FUNCTION_BLOCK KukaRobot
VAR_INPUT
END_VAR
VAR
	wSendData : DWORD;
END_VAR
VAR_OUTPUT
	wOutputWord AT %Q* : DWORD;
END_VAR

METHOD SendData : BOOL
VAR_INPUT
	bFailure : BOOL := FALSE;
END_VAR
IF bFailure THEN
	wOutputWord := 16#00000001;
ELSE
	wOutputWord:= 16#00000000;
END_IF
END_METHOD

END_FUNCTION_BLOCK

(* stored: Version 1.1.0.1, ProductVersion 3.1.4024.12
   POU KukaRobot: Id {468c34ef-d238-4a9f-8ae3-3cdce425a776}, SpecialFunc None
   Method SendData: Id {b33c5007-83ac-428f-b48d-44026c54e9d4} *)
